// TIA Portal V18 export
FUNCTION_BLOCK "MD"   // FB11, FBD
{ S7_Optimized_Access := 'TRUE' }
VERSION : 0.1
// stored: AutoNumber true, IsIECCheckEnabled false, IsRetainMemResEnabled false, MemoryReserve 100, SetENOAutomatically false, UDAEnableTagReadback false
   VAR_OUTPUT
      CHAN_TR : Bool;
   END_VAR
   VAR_IN_OUT
      AUT : Bool;
      MAN : Bool := true;
      SERV : Bool;
   END_VAR
   VAR
      lbs { S7_SetPoint := 'True'} : "last_button_stands";
   END_VAR
BEGIN

REGION Network 1
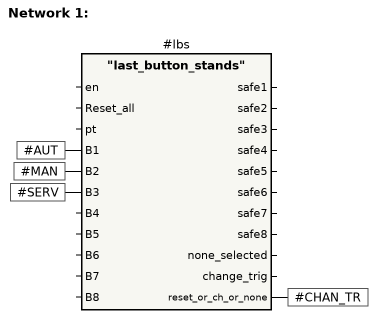
   #lbs(B1 := #AUT, B2 := #MAN, B3 := #SERV, reset_or_ch_or_none => #CHAN_TR);   // "last_button_stands"
END_REGION
END_FUNCTION_BLOCK
